Fanuc KAREL source: kt00538.KL

-- PROVISIONAL review KL for V1013-1; original PC SHA256 c4dc886e29dc8becd8bd4e9b29c59002a6033d02e6a5723d7cd0b7212e1a2bab
-- Incomplete behavior may be omitted. Consult companion uncertainty JSON. Do not deploy.
PROGRAM KT00538
%NOLOCKGROUP
VAR
  OUT : BOOLEAN
-- UNRESOLVED_DECL P1 type=000199
-- UNRESOLVED_DECL P2 type=000102
BEGIN
  -- UNRESOLVED_PC offsets 5-20; opcodes 2E,22,32,35
  -- UNRESOLVED_PC offsets 25-58; opcodes 49,7E,49,7E,AC,23
  -- UNRESOLVED_PC offsets 63-67; opcodes 7F
END KT00538
